(* IEC 61131-3 sources: LabBench/POU/02_Equipments, 1 file *)

(* ---- PRG_EquipmentProcessing.st ---- *)
(*==============================================================================
    Название:    PRG_EquipmentProcessing
    Автор:       Редько А.
    Дата:        2025-04-27
    Версия:      1.0

    Описание:    Программа управления оборудованием стенда
==============================================================================*)
PROGRAM PRG_EquipmentProcessing
VAR
    (* Экземпляры функциональных блоков *)
    fbPropValve: FB_PropValve;    (* Пропорциональный кран *)
    fbEMValve: FB_EMValve;        (* Электромагнитный клапан *)

    (* Локальные переменные *)
    bEmergencyStop: BOOL := FALSE; (* Общий сигнал аварийного останова *)
END_VAR

(* ======================================================================== *)
(* Обработка общих сигналов для всех устройств                              *)
(* ======================================================================== *)

(* Проверка общего сигнала аварийного останова *)
(* Здесь можно добавить логику для определения аварийных ситуаций *)

(* ======================================================================== *)
(* Управление пропорциональным краном                                       *)
(* ======================================================================== *)

(* Установка внешней команды аварийного останова *)
stPropValve.stCommands.bExtEmergencyStop := bEmergencyStop;

(* Вызов функционального блока *)
fbPropValve(
    stValve := stPropValve,
    rFeedbackSignal := AI_Position_PropValve,  (* Сигнал уже масштабирован в конфигурации *)
    bEnable := TRUE,
    rControlSignal => AO_SetPosition_PropValve
);

(* ======================================================================== *)
(* Управление электромагнитным клапаном                                     *)
(* ======================================================================== *)

(* Обновление порога предупреждения из SCADA *)
stEMValve.tWarningThreshold := GVL_in_SCADA_EMValve_WarningTime; (* Порог предупреждения *)

(* Вызов функционального блока *)
fbEMValve(
    stValve := stEMValve,
    bManualOpenCommand := GVL_in_SCADA_EMValve_Open,   (* Команда открытия в ручном режиме *)
    bAutoOpenCommand := GVL_in_SCADA_EMValve_AutoOpen, (* Команда открытия от регулятора *)
    bEmergencyStop := bEmergencyStop,               (* Общий сигнал аварийного останова *)
    eMode := GVL_in_SCADA_EMValve_Mode,              (* Режим работы электромагнитного клапана *)
    bEnable := TRUE,
    bOutputSignal => DO_Open_Valve
);
